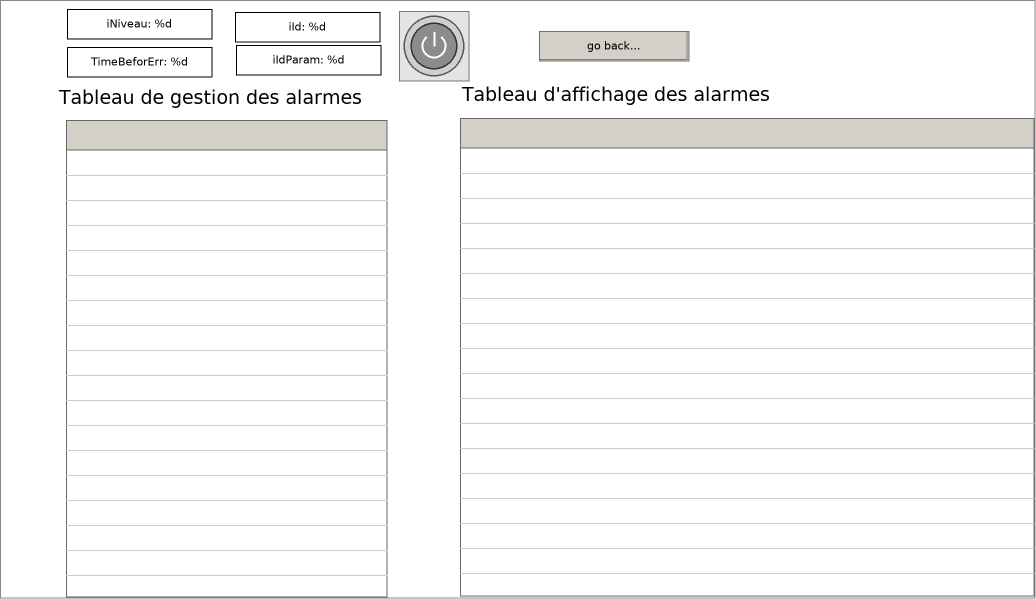
VISUALIZATION Vi_Alarmes  // 1036x599
    Table (66,120 321x477), data array: fbErrorAdmin.stActError
        p3854506369: fbErrorAdmin.stActError[INDEX].iId
        p1892666644: fbErrorAdmin.stActError[INDEX].iParam
        p338671338: fbErrorAdmin.stActError[INDEX].iIndexOrigine
        p2170511999: fbErrorAdmin.stActError[INDEX].iLevel
    Label (56,77 342x41), "Tableau de gestion des alarmes"
    Label (459,74 342x41), "Tableau d'affichage des alarmes"
    Table (460,118 574x478), data array: fbErrorViewer.astErrorView
        p3854506369: fbErrorViewer.astErrorView[INDEX].id
        p1892666644: fbErrorViewer.astErrorView[INDEX].idparam
        p338671338: fbErrorViewer.astErrorView[INDEX].sMess
    Rectangle (67,9 145x30), "iNiveau: %d", text variable: MAIN.iNiveau
        OnMouseClick: write the text variable via Default
    Rectangle (67,47 145x30), "TimeBeforErr: %d", text variable: MAIN.TimeBeforError
        OnMouseClick: write the text variable via Default
    Rectangle (235,12 145x30), "iId: %d", text variable: MAIN.iId
        OnMouseClick: write the text variable via Default
    Rectangle (236,45 145x30), "iIdParam: %d", text variable: MAIN.iIdParam
        OnMouseClick: write the text variable via Default
    PowerSwitch (399,11 70x70), variable: MAIN.xSetError, behaviour: TAP, style: Switch-PowerSwitch-Gray
    Button (539,31 150x30), "go back..."
        OnMouseClick: change screen: Visualization
END_VISUALIZATION

(* stored: Version 1.1.0.1, ProductVersion 3.1.4020.6
   Visu Vi_Alarmes: Id {cad58a7a-4682-40d7-b457-faf9138f2228} *)
